(* CoDeSys 2.3 library: TcBaseMath.lib *)

(* POU FW_Floor, ST *)
FUNCTION FW_Floor 	: 	LREAL
VAR_INPUT
	lr_in			:	LREAL;
END_VAR
VAR
END_VAR
;
END_FUNCTION

(* POU FW_LrealFrac, ST *)
FUNCTION FW_LrealFrac 	: 	LREAL
VAR_INPUT
	lr_in			:	LREAL;
END_VAR
VAR
END_VAR
;
END_FUNCTION

(* POU FW_LrealModP, ST *)
FUNCTION FW_LrealModP 	: 	LREAL
VAR_INPUT
	lr_val			:	LREAL;
	lr_mod 			: LREAL;
END_VAR
VAR
END_VAR
;
END_FUNCTION

(* POU FW_LrealTrunc, ST *)
FUNCTION FW_LrealTrunc 	: 	LREAL
VAR_INPUT
	lr_in			:	LREAL;
END_VAR
VAR
END_VAR
;
END_FUNCTION
